# EPICS autosave request: galilDmc30017App/Db/galil_dmc30017_digital_in_4_7.req
# The files listed here are located at <GALIL support top>/GalilSup/Db
# as they are provided by the Galil Support Module

# Digital input bits 4-7
file "galil_digital_in_bit.req" P=$(P), R=$(DIG_IN4)
file "galil_digital_in_bit.req" P=$(P), R=$(DIG_IN5)
file "galil_digital_in_bit.req" P=$(P), R=$(DIG_IN6)
file "galil_digital_in_bit.req" P=$(P), R=$(DIG_IN7)
